ABB RobotStudio station: Assgnt_2_Final.rspag

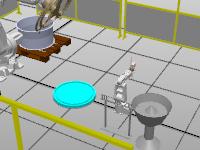
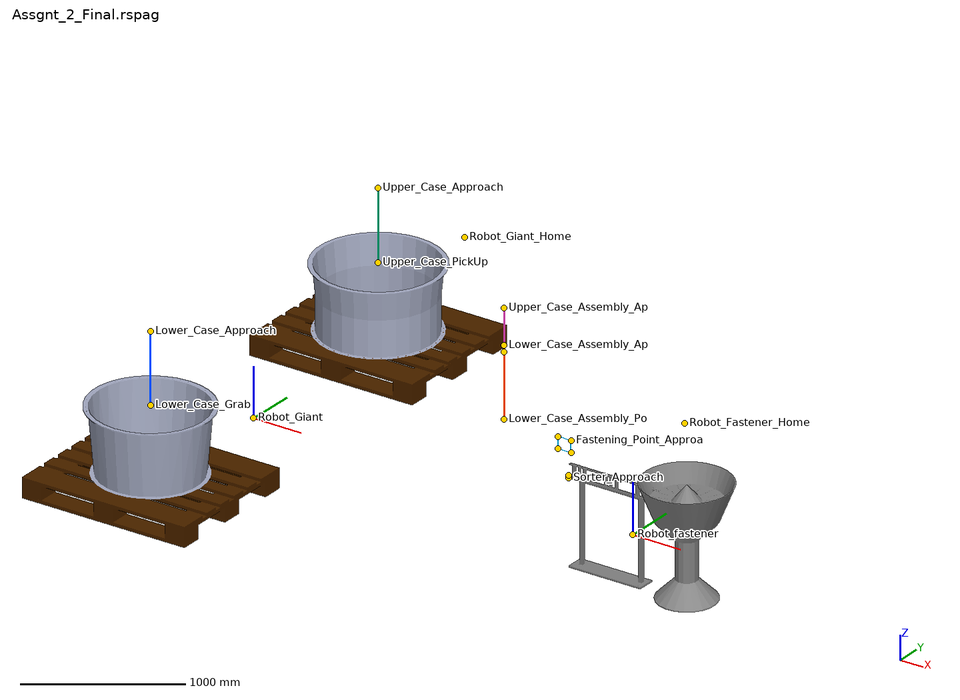
[picture v1: parts stored in the station drawn from their meshes, with robot base, taught points and paths (robot models come from the ABB library and are not in the file)]
--- station ---
Station Assign2_Final (saved by RobotStudio 21.2.9526.0)
Controller Sync_Controller
  mechanical unit ROB_1: Robot_Giant, 6 joints, base frame (0, 0, 0) mm
  mechanical unit ROB_2: Robot_fastener, 6 joints, base frame (2800, 0, 0) mm, rotated rx 0 ry 0 rz 180 deg
Layout (positions relative to the parent item):
  - Robot_Giant [mechanism, from Robots\IRB6620_150_220_G_01.rslib] at (0, 0, 0) mm; joint values [0, 0, 0, 0, 0.5236, 0] (rad or m)
  - UpperEngineCase [part] at (80, 1200, 136) mm, size 855.3 x 860 x 451.6 mm
  - M8_Lock_Nut [part] at (3456.05, -671.29, 653.31) mm, size 15.6 x 13.7 x 11 mm
  - Bolt_nothread [part] at (3473.13, -433.44, 655.7) mm, rotated rx -82.72 ry 0 rz 0 deg, size 20 x 20 x 36 mm
  - Rotating_Base_Mech [mechanism, from Libraries\Rotating_Base_Mech.rslib] at (1850, 0, 0) mm, rotated rx 0 ry 0 rz 37.5 deg; joint values [0] (rad or m)
  - Fence_2500_V1_2 [graphiccomponentgroup, from Equipment\Fence_2500.rslib] at (4110.06, 2559.49, 0) mm, rotated rx 0 ry 0 rz 90 deg
    - Body 1 [part, from Equipment\Fence_2500.rslib]
    - Body 2 [part, from Equipment\Fence_2500.rslib]
  - Fence_2500_H2_2 [graphiccomponentgroup, from Equipment\Fence_2500.rslib] at (-1516.69, -2535.36, 0) mm
    - Body 1 [part, from Equipment\Fence_2500.rslib]
    - Body 2 [part, from Equipment\Fence_2500.rslib]
  - Fence_2500_V1 [graphiccomponentgroup, from Equipment\Fence_2500.rslib] at (1527.78, 2566.59, 0) mm, rotated rx 0 ry 0 rz 90 deg
    - Body 1 [part, from Equipment\Fence_2500.rslib]
    - Body 2 [part, from Equipment\Fence_2500.rslib]
  - Fence_2500_V2 [graphiccomponentgroup, from Equipment\Fence_2500.rslib] at (1521.75, -2665.51, 0) mm, rotated rx 0 ry 0 rz 90 deg
    - Body 1 [part, from Equipment\Fence_2500.rslib]
    - Body 2 [part, from Equipment\Fence_2500.rslib]
  - Fence_2500_H1_2 [graphiccomponentgroup, from Equipment\Fence_2500.rslib] at (4779.67, -2566.91, 0) mm
    - Body 1 [part, from Equipment\Fence_2500.rslib]
    - Body 2 [part, from Equipment\Fence_2500.rslib]
  - Fence_2500_V2_2 [graphiccomponentgroup, from Equipment\Fence_2500.rslib] at (4153.21, -2654.07, 0) mm, rotated rx 0 ry 0 rz 90 deg
    - Body 1 [part, from Equipment\Fence_2500.rslib]
    - Body 2 [part, from Equipment\Fence_2500.rslib]
  - Fence_2500_H1 [graphiccomponentgroup, from Equipment\Fence_2500.rslib] at (4775.16, 0, 0) mm
    - Body 1 [part, from Equipment\Fence_2500.rslib]
    - Body 2 [part, from Equipment\Fence_2500.rslib]
  - Fence_2500_H2 [graphiccomponentgroup, from Equipment\Fence_2500.rslib] at (-1486.79, 0, 0) mm
    - Body 1 [part, from Equipment\Fence_2500.rslib]
    - Body 2 [part, from Equipment\Fence_2500.rslib]
  - Pallet_1 [part] at (80, -1200, 138) mm, rotated rx 90 ry 0 rz 0 deg, size 1200 x 138 x 1000 mm
  - Pallet_2 [part] at (80, 1200, 138) mm, rotated rx 90 ry 0 rz 0 deg, size 1200 x 138 x 1000 mm
  - Robot_fastener [mechanism, from Robots\IRB120_3_58_G_01.rslib] at (2800, 0, 0) mm, rotated rx 0 ry 0 rz 180 deg; joint values [-1.5708, 0, 0, 0, 0, 0] (rad or m)
  - IRC5_Control-Module [part, from Equipment\IRC5_Control-Module.rslib] at (-932.79, 0, 100) mm, rotated rx 90 ry 0 rz 90 deg
  - SC_Grabber [smart component, from Libraries\SC_Grabber.rslib] at (1380.21, 0, 1755) mm, rotated rx 180 ry 60 rz 180 deg
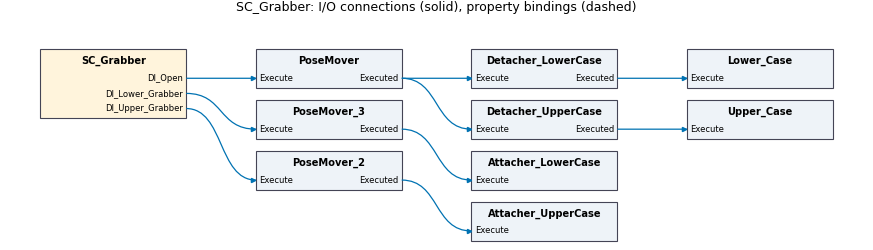
      connections:
        SC_Grabber.DI_Open -> PoseMover.Execute
        SC_Grabber.DI_Lower_Grabber -> PoseMover_3.Execute
        SC_Grabber.DI_Upper_Grabber -> PoseMover_2.Execute
        PoseMover_2.Executed -> Attacher_UpperCase.Execute
        PoseMover_3.Executed -> Attacher_LowerCase.Execute
        PoseMover.Executed -> Detacher_LowerCase.Execute
        PoseMover.Executed -> Detacher_UpperCase.Execute
        Detacher_LowerCase.Executed -> Lower_Case.Execute
        Detacher_UpperCase.Executed -> Upper_Case.Execute
    - Mech_Grabber [mechanism, from Libraries\SC_Grabber.rslib] at (0, 0, 0) mm; joint values [0, 0, 0] (rad or m)
    - PoseMover [smart component, from Components\PoseMover.rslib]
        properties: Mechanism=Mech_Grabber; Pose=2; Duration=0.5
    - PoseMover_2 [smart component, from Components\PoseMover.rslib]
        properties: Mechanism=Mech_Grabber; Pose=3; Duration=0.5
    - PoseMover_3 [smart component, from Components\PoseMover.rslib]
        properties: Mechanism=Mech_Grabber; Pose=4; Duration=0.5
    - Attacher_LowerCase [smart component, from Components\Attacher.rslib]
        properties: Parent=Mech_Grabber; Flange=0; Child=LowerEngineCase; Mount=false; Offset=[0 0 0]; Orientation=[0 0 0]
    - Attacher_UpperCase [smart component, from Components\Attacher.rslib]
        properties: Parent=Mech_Grabber; Flange=0; Child=UpperEngineCase; Mount=false; Offset=[0 0 0]; Orientation=[0 0 0]
    - Detacher_LowerCase [smart component, from Components\Detacher.rslib]
        properties: Child=LowerEngineCase; KeepPosition=true
    - Detacher_UpperCase [smart component, from Components\Detacher.rslib]
        properties: Child=UpperEngineCase; KeepPosition=true
    - Lower_Case [smart component, from Components\SetParent.rslib]
        properties: Child=LowerEngineCase; Parent=Rotating_Base_Mech; KeepTransform=true
    - Upper_Case [smart component, from Components\SetParent.rslib]
        properties: Child=UpperEngineCase; Parent=Rotating_Base_Mech; KeepTransform=true
  - New Nut and Bolt Sorter [part] at (3000, -525, 0) mm, size 1163.5 x 597 x 775 mm
  - SC_Nut_Bolt_Sorter [smart component, from Libraries\SC_Nut_Bolt_Sorter.rslib]
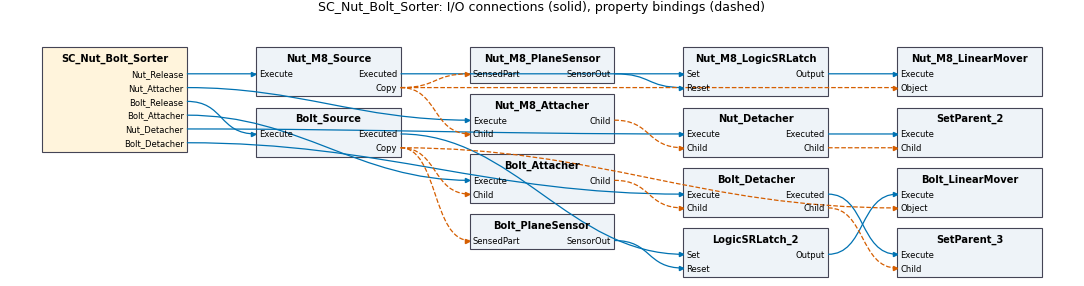
      connections:
        SC_Nut_Bolt_Sorter.Nut_Release -> Nut_M8_Source.Execute
        Nut_M8_Source.Executed -> Nut_M8_LogicSRLatch.Set
        Nut_M8_PlaneSensor.SensorOut -> Nut_M8_LogicSRLatch.Reset
        Nut_M8_LogicSRLatch.Output -> Nut_M8_LinearMover.Execute
        SC_Nut_Bolt_Sorter.Nut_Attacher -> Nut_M8_Attacher.Execute
        SC_Nut_Bolt_Sorter.Bolt_Release -> Bolt_Source.Execute
        Bolt_Source.Executed -> LogicSRLatch_2.Set
        LogicSRLatch_2.Output -> Bolt_LinearMover.Execute
        Bolt_PlaneSensor.SensorOut -> LogicSRLatch_2.Reset
        SC_Nut_Bolt_Sorter.Bolt_Attacher -> Bolt_Attacher.Execute
        SC_Nut_Bolt_Sorter.Nut_Detacher -> Nut_Detacher.Execute
        SC_Nut_Bolt_Sorter.Bolt_Detacher -> Bolt_Detacher.Execute
        Nut_Detacher.Executed -> SetParent_2.Execute
        Bolt_Detacher.Executed -> SetParent_3.Execute
        Nut_M8_Source.Copy => Nut_M8_LinearMover.Object
        Bolt_Source.Copy => Bolt_LinearMover.Object
        Nut_M8_Attacher.Child => Nut_Detacher.Child
        Bolt_Attacher.Child => Bolt_Detacher.Child
        Nut_M8_Source.Copy => Nut_M8_PlaneSensor.SensedPart
        Bolt_Source.Copy => Bolt_PlaneSensor.SensedPart
        Nut_M8_Source.Copy => Nut_M8_Attacher.Child
        Bolt_Source.Copy => Bolt_Attacher.Child
        Nut_Detacher.Child => SetParent_2.Child
        Bolt_Detacher.Child => SetParent_3.Child
    - Nut_M8_Source [smart component, from Components\Source.rslib]
        properties: Source=M8_Lock_Nut; Copy=(none); Parent=(none); Position=[3.340616 -0.525502 0.575]; Orientation=[0 0 0]; Transient=false; PhysicsBehavior=0
    - Nut_M8_LogicSRLatch [smart component, from Components\LogicSRLatch.rslib]
    - Nut_M8_PlaneSensor [smart component, from Components\PlaneSensor.rslib]
        properties: Origin=[2.69 -0.58 0.55]; Axis1=[0 0.1 0]; Axis2=[0 0 0.06]; SensedPart=(none)
      - _sensorPart_ [part, from Libraries\SC_Nut_Bolt_Sorter.rslib]
    - Nut_M8_LinearMover [smart component, from Components\LinearMover.rslib]
        properties: Object=(none); Direction=[-0.64172 0 0]; Speed=0.3; Reference=Global; ReferenceObject=(none)
    - Nut_M8_Attacher [smart component, from Components\Attacher.rslib]
        properties: Parent=SC_Fastener_New; Flange=0; Child=(none); Mount=false; Offset=[0 0 0]; Orientation=[0 0 0]
    - Bolt_Attacher [smart component, from Components\Attacher.rslib]
        properties: Parent=SC_Fastener_New; Flange=0; Child=(none); Mount=false; Offset=[0 0 0]; Orientation=[0 0 0]
    - Bolt_LinearMover [smart component, from Components\LinearMover.rslib]
        properties: Object=(none); Direction=[-1 0 0]; Speed=0.3; Reference=Global; ReferenceObject=(none)
    - Bolt_PlaneSensor [smart component, from Components\PlaneSensor.rslib]
        properties: Origin=[2.69 -0.58 0.65]; Axis1=[0 0.1 0]; Axis2=[0 0 0.06]; SensedPart=(none)
      - _sensorPart_ [part, from Libraries\SC_Nut_Bolt_Sorter.rslib]
    - LogicSRLatch_2 [smart component, from Components\LogicSRLatch.rslib]
    - Bolt_Source [smart component, from Components\Source.rslib]
        properties: Source=Bolt_nothread; Copy=(none); Parent=(none); Position=[3.306216 -0.525502 0.64]; Orientation=[0 0 0]; Transient=false; PhysicsBehavior=0
    - Nut_Detacher [smart component, from Components\Detacher.rslib]
        properties: Child=(none); KeepPosition=true
    - Bolt_Detacher [smart component, from Components\Detacher.rslib]
        properties: Child=(none); KeepPosition=true
    - SetParent_2 [smart component, from Components\SetParent.rslib]
        properties: Child=(none); Parent=Rotating_Base_Mech; KeepTransform=true
    - SetParent_3 [smart component, from Components\SetParent.rslib]
        properties: Child=(none); Parent=Rotating_Base_Mech; KeepTransform=true
  - LowerEngineCase [part] at (80, -1200, 136) mm, size 821.5 x 826 x 454 mm
  - SC_Fastener_New [smart component, from Libraries\SC_Fastener_New.rslib] at (2800, 374, 630) mm, rotated rx 0 ry 90 rz 90 deg
      connections:
        SC_Fastener_New.FNDI_Home -> PoseMover.Execute
        SC_Fastener_New.FNDI_Open -> PoseMover_2.Execute
        SC_Fastener_New.FNDI_ClosePick -> PoseMover_3.Execute
    - Mech_Fastening_New [mechanism, from Libraries\SC_Fastener_New.rslib] at (0, 0, 0) mm; joint values [-0.07, 0.0705] (rad or m)
    - PoseMover [smart component, from Components\PoseMover.rslib]
        properties: Mechanism=Mech_Fastening_New; Pose=1; Duration=0.5
    - PoseMover_2 [smart component, from Components\PoseMover.rslib]
        properties: Mechanism=Mech_Fastening_New; Pose=2; Duration=0.5
    - PoseMover_3 [smart component, from Components\PoseMover.rslib]
        properties: Mechanism=Mech_Fastening_New; Pose=3; Duration=0.5
  - SC_Rotate_Base [smart component, from Libraries\SC_Rotate_Base.rslib]
      connections:
        SC_Rotate_Base.DI_Rotate -> Base.Execute
    - Base [smart component, from Components\Rotator2.rslib]
        properties: Object=Rotating_Base_Mech; CenterPoint=[0 0 0]; Axis=[0 0 0.001]; Angle=0.130899693899575; Duration=1; Reference=Local; ReferenceObject=(none)
Attachment: SC_Grabber is attached to Robot_Giant / Link6
Attachment: SC_Fastener_New is attached to Robot_fastener / Link6
Station signals: DI Trail_Breaker
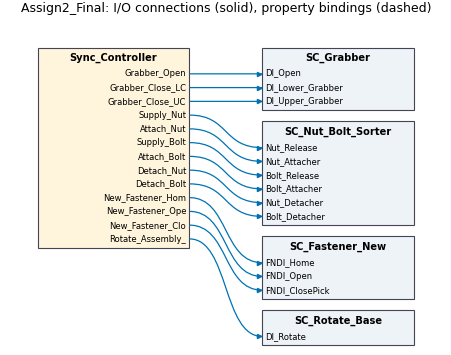
Station logic (signal -> signal, property => property):
  Sync_Controller.Grabber_Open -> SC_Grabber.DI_Open
  Sync_Controller.Grabber_Close_LC -> SC_Grabber.DI_Lower_Grabber
  Sync_Controller.Grabber_Close_UC -> SC_Grabber.DI_Upper_Grabber
  Sync_Controller.Supply_Nut -> SC_Nut_Bolt_Sorter.Nut_Release
  Sync_Controller.Attach_Nut -> SC_Nut_Bolt_Sorter.Nut_Attacher
  Sync_Controller.Supply_Bolt -> SC_Nut_Bolt_Sorter.Bolt_Release
  Sync_Controller.Attach_Bolt -> SC_Nut_Bolt_Sorter.Bolt_Attacher
  Sync_Controller.Detach_Nut -> SC_Nut_Bolt_Sorter.Nut_Detacher
  Sync_Controller.Detach_Bolt -> SC_Nut_Bolt_Sorter.Bolt_Detacher
  Sync_Controller.New_Fastener_Home -> SC_Fastener_New.FNDI_Home
  Sync_Controller.New_Fastener_Open -> SC_Fastener_New.FNDI_Open
  Sync_Controller.New_Fastener_ClosePick -> SC_Fastener_New.FNDI_ClosePick
  Sync_Controller.Rotate_Assembly_Base -> SC_Rotate_Base.DI_Rotate

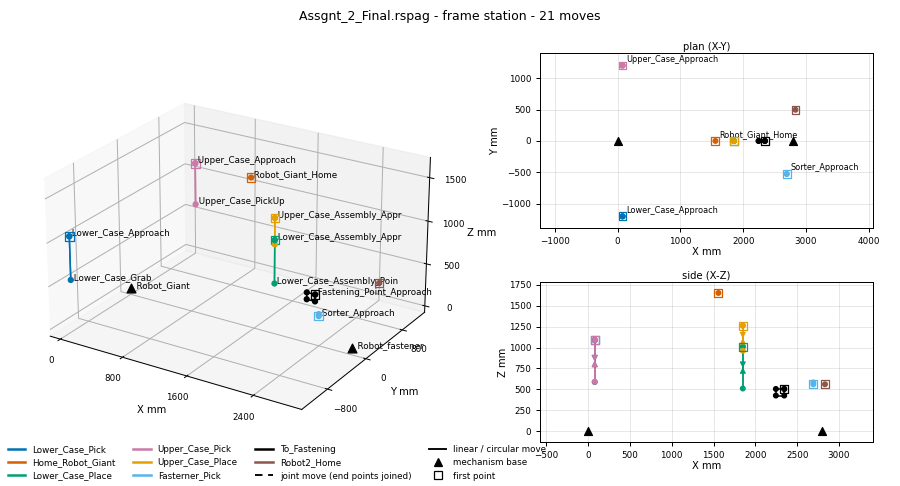
[picture p0: tool path of Assgnt_2_Final.rspag in frame station, 21 of 21 moves have a stored position in this frame; points joined in program order, loops and branches not executed]
--- Backups/Sync_Controller/RAPID/TASK1/PROGMOD/CalibData.mod ---
MODULE CalibData
    PERS tooldata Mech_Grabber_1:=[TRUE,[[0,0,205.5],[1,0,0,0]],[2,[0,0,200],[1,0,0,0],0,0,0]];
    TASK PERS wobjdata Wobj_Lower_Case:=[FALSE,TRUE,"",[[80.0405,-1200,592],[0.999974,-0.00506277,0.00506303,0.000025634]],[[0,0,0],[1,0,0,0]]];
    TASK PERS wobjdata Wobj_Upper_Case:=[FALSE,TRUE,"",[[80,1200,589.619],[1,0,0,0]],[[0,0,0],[1,0,0,0]]];
    TASK PERS wobjdata Wobj_Assembly:=[FALSE,TRUE,"",[[1850,0,60],[1,0,0,0]],[[0,0,0],[1,0,0,0]]];
ENDMODULE

--- Backups/Sync_Controller/RAPID/TASK1/PROGMOD/Module1.mod ---
MODULE Module1
        CONST robtarget Lower_Case_Approach:=[[-5.063031994,-5.022012339,495.949144175],[-0.000000184,0.707106781,0.707070529,0.007160025],[0,0,0,0],[9E+09,9E+09,9E+09,9E+09,9E+09,9E+09]];
    CONST robtarget Lower_Case_Grab:=[[0.000000003,0.0405001,-3.999589872],[0.000000184,0.707106781,0.707070529,0.007160025],[0,0,0,0],[9E+09,9E+09,9E+09,9E+09,9E+09,9E+09]];
    CONST robtarget Robot_Giant_Home:=[[1558.173301235,0,1652.25],[0.5,0,0.866025404,0],[0,0,0,0],[9E+09,9E+09,9E+09,9E+09,9E+09,9E+09]];
    CONST robtarget Lower_Case_Assembly_Approach:=[[0,0,950],[0,0,1,0],[0,0,0,0],[9E+09,9E+09,9E+09,9E+09,9E+09,9E+09]];
    CONST robtarget Lower_Case_Assembly_Point:=[[0,0,450],[0,0,1,0],[0,0,0,0],[9E+09,9E+09,9E+09,9E+09,9E+09,9E+09]];
    CONST robtarget Upper_Case_Approach:=[[0,0,500],[0,-0.707106779,0.707106783,-0.000000368],[0,0,0,0],[9E+09,9E+09,9E+09,9E+09,9E+09,9E+09]];
    CONST robtarget Upper_Case_PickUp:=[[0,0,0],[0,-0.707106779,0.707106783,-0.000000368],[0,-1,-1,0],[9E+09,9E+09,9E+09,9E+09,9E+09,9E+09]];
    CONST robtarget Upper_Case_Assembly_Approach:=[[0,0,1201.62],[0,0,1,0],[0,0,0,0],[9E+09,9E+09,9E+09,9E+09,9E+09,9E+09]];
    CONST robtarget Upper_Case_Assembly_Point:=[[0,0,901.62],[0,0,1,0],[0,0,0,0],[9E+09,9E+09,9E+09,9E+09,9E+09,9E+09]];
!***********************************************************
    !
    ! Module:  Module1
    !
    ! Description:
    !   <Insert description here>
    !
    ! Author: Santosh Govindaraj
    !
    ! Version: 1.0
    !
    !***********************************************************


    !***********************************************************
    !
    ! Procedure main
    !
    !   This is the entry point of your program
    !
    !***********************************************************
    PROC main()
        !Add your code here
        Home_Robot_Giant;
        Lower_Case_Pick;
        Lower_Case_Place;
        Upper_Case_Pick;
        Upper_Case_Place;
        Home_Robot_Giant;
    ENDPROC
    PROC Lower_Case_Pick()
        SetDO Grabber_Open,1;
        SetDO Grabber_Close_LC,0;
        MoveL Lower_Case_Approach,v1000,z100,Mech_Grabber_1\WObj:=Wobj_Lower_Case;
        MoveL Lower_Case_Grab,v1000,z100,Mech_Grabber_1\WObj:=Wobj_Lower_Case;
        WaitTime 0.5;
        SetDO Grabber_Open,0;
        SetDO Grabber_Close_LC,1;
        WaitTime 1;
        MoveL Lower_Case_Approach,v1000,z100,Mech_Grabber_1\WObj:=Wobj_Lower_Case;
    ENDPROC
    PROC MAIN_ROB1()
        Home_Robot_Giant;
        Lower_Case_Pick;
        Lower_Case_Place;
        Upper_Case_Pick;
        Upper_Case_Place;
        Home_Robot_Giant;
    ENDPROC
    PROC Home_Robot_Giant()
        MoveL Robot_Giant_Home,v1000,z100,Mech_Grabber_1\WObj:=wobj0;
    ENDPROC
    PROC Lower_Case_Place()
        MoveL Lower_Case_Assembly_Approach,v1000,z100,Mech_Grabber_1\WObj:=Wobj_Assembly;
        MoveL Lower_Case_Assembly_Point,v1000,z100,Mech_Grabber_1\WObj:=Wobj_Assembly;
        SetDO Grabber_Close_LC,0;
        WaitTime 1;
        SetDO Grabber_Open,1;
        SetDO Grabber_Open,0;
        WaitTime 1;
        MoveL Lower_Case_Assembly_Approach,v1000,z100,Mech_Grabber_1\WObj:=Wobj_Assembly;
    ENDPROC
    PROC Upper_Case_Pick()
        SetDO Grabber_Open,1;
        SetDO Grabber_Close_UC,0;
        SetDO Grabber_Open,0;
        MoveL Upper_Case_Approach,v1000,z100,Mech_Grabber_1\WObj:=Wobj_Upper_Case;
        MoveL Upper_Case_PickUp,v1000,z100,Mech_Grabber_1\WObj:=Wobj_Upper_Case;
        WaitTime 0.5;
        SetDO Grabber_Close_UC,1;
        WaitTime 1;
        MoveL Upper_Case_Approach,v1000,z100,Mech_Grabber_1\WObj:=Wobj_Upper_Case;
    ENDPROC
    PROC Upper_Case_Place()
        MoveL Upper_Case_Assembly_Approach,v1000,z100,Mech_Grabber_1\WObj:=Wobj_Assembly;
        MoveL Upper_Case_Assembly_Point,v1000,z100,Mech_Grabber_1\WObj:=Wobj_Assembly;
        SetDO Grabber_Close_UC,0;
        WaitTime 1;
        SetDO Grabber_Open,1;
        SetDO Grabber_Open,0;
        WaitTime 1;
        MoveL Upper_Case_Assembly_Approach,v1000,z100,Mech_Grabber_1\WObj:=Wobj_Assembly;
    ENDPROC
    PROC Path_10()

    ENDPROC
    PROC ROBOT()
        Home_Robot_Giant;
        Lower_Case_Pick;
        Lower_Case_Place;
        Upper_Case_Pick;
        Upper_Case_Place;
        Home_Robot_Giant;
    ENDPROC
ENDMODULE

--- Backups/Sync_Controller/RAPID/TASK2/PROGMOD/CalibData.mod ---
MODULE CalibData
    PERS tooldata Mech_Fastener_1:=[TRUE,[[-12,-31.5,121],[1,0,0,0]],[1,[0.1,0,0],[1,0,0,0],0,0,0]];
    PERS tooldata Mech_Fastner_1:=[TRUE,[[69,-32,122],[0.707107,0,0.707107,0]],[1.5,[0.1,0,0],[1,0,0,0],0,0,0]];
    TASK PERS wobjdata Wobj_Sorter:=[FALSE,TRUE,"",[[2699.22,-537.502,584],[1,0,0,0]],[[0,0,0],[1,0,0,0]]];
    TASK PERS wobjdata Wobj_Fastening:=[FALSE,TRUE,"",[[1850,0,60],[1,0,0,0]],[[0,0,0],[1,0,0,0]]];
    PERS tooldata Mech_Fastening_New_1:=[TRUE,[[139.999,-31.395,121.281],[0.707107,0,0.707107,0]],[2,[50,50,50],[1,0,0,0],0,0,0]];
ENDMODULE

--- Backups/Sync_Controller/RAPID/TASK2/PROGMOD/Module1.mod ---
MODULE Module1
        CONST robtarget Target_10:=[[2831.999489549,496.000032596,560.999998333],[0.000000002,0.707107145,-0.707106417,0.000000002],[-1,0,-1,0],[9E+09,9E+09,9E+09,9E+09,9E+09,9E+09]];
    CONST robtarget Target_20:=[[2742.402,-523,589.664],[0.000000002,0.707106417,0.707107145,0.000000002],[0,-2,1,1],[9E+09,9E+09,9E+09,9E+09,9E+09,9E+09]];
    CONST robtarget Target_30:=[[2745.508,-494.542,588.187],[0.000000002,0.707106417,0.707107145,0.000000002],[0,-2,1,1],[9E+09,9E+09,9E+09,9E+09,9E+09,9E+09]];
    CONST robtarget Bolt_attac:=[[2745.875,-494.542,676],[0.000000002,0.707106417,0.707107145,0.000000002],[0,0,-1,0],[9E+09,9E+09,9E+09,9E+09,9E+09,9E+09]];
    CONST robtarget Sorter_Approach:=[[-6.6,12,-24],[0,0.707106781,0.707106781,0],[0,0,-1,0],[9E+09,9E+09,9E+09,9E+09,9E+09,9E+09]];
    CONST robtarget Sorter_Pick:=[[-6.6,12,-2],[0,0.707106781,0.707106781,0],[0,0,-1,0],[9E+09,9E+09,9E+09,9E+09,9E+09,9E+09]];
    CONST robtarget Fastening_Point_Approach:=[[495,0,445],[0,1,0,0],[0,-2,1,0],[9E+09,9E+09,9E+09,9E+09,9E+09,9E+09]];
    CONST robtarget Fastening_Point:=[[395,0,445],[0,1,0,0],[0,-2,1,0],[9E+09,9E+09,9E+09,9E+09,9E+09,9E+09]];
    CONST robtarget Robot_Fastener_Home:=[[2831.999489549,496.000032596,560.999998333],[0.000000002,0.707107145,-0.707106417,0.000000002],[-1,0,-1,0],[9E+09,9E+09,9E+09,9E+09,9E+09,9E+09]];
    CONST robtarget Fastening_Point_Down:=[[395,0,366],[0,1,0,0],[0,-2,1,0],[9E+09,9E+09,9E+09,9E+09,9E+09,9E+09]];
    CONST robtarget Fastening_Wait_For_Next:=[[495,0,366],[0,1,0,0],[0,-2,1,0],[9E+09,9E+09,9E+09,9E+09,9E+09,9E+09]];
!***********************************************************
    !
    ! Module:  Module1
    !
    ! Description:
    !   <Insert description here>
    !
    ! Author: Santosh Govindaraj
    !
    ! Version: 1.0
    !
    !***********************************************************


    !***********************************************************
    !
    ! Procedure main
    !
    !   This is the entry point of your program
    !
    !***********************************************************
    PROC main()
        !Add your code here
    ENDPROC
    PROC Suppliers()
        SetDO Supply_Nut,0;
        SetDO Supply_Bolt,0;
        WaitTime 0.5;
        SetDO Supply_Nut,1;
        SetDO Supply_Bolt,1;
        WaitTime 1;
    ENDPROC
    PROC Robot2_Task()
        SetDO New_Fastener_Home,0;
        WaitTime 18;
        Robot2_Home;
        FOR loop FROM 0 TO 47 DO
            Fasten_And_Rotate;
        ENDFOR
        Robot2_Home;
    ENDPROC
    PROC Fasterner_Pick()
        SetDO New_Fastener_Open,1;
        SetDO New_Fastener_Open,0;
        SetDO Attach_Nut,0;
        SetDO Attach_Bolt,0;
        WaitTime 0.5;
        MoveJ Sorter_Approach,v2000,fine,Mech_Fastening_New_1\WObj:=Wobj_Sorter;
        MoveL Sorter_Pick,v1000,fine,Mech_Fastening_New_1\WObj:=Wobj_Sorter;
        SetDO Attach_Nut,1;
        SetDO New_Fastener_ClosePick,1;
        WaitTime 0.5;
        SetDO New_Fastener_ClosePick,0;
        SetDO Attach_Bolt,1;
        WaitTime 0.5;
        SetDO Attach_Nut,0;
        SetDO Attach_Bolt,0;
    ENDPROC
    PROC To_Fastening()
        MoveJ Fastening_Point_Approach,v1000,fine,Mech_Fastening_New_1\WObj:=Wobj_Fastening;
        MoveJ Fastening_Point,v500,fine,Mech_Fastening_New_1\WObj:=Wobj_Fastening;
        WaitTime 0.5;
        SetDO Detach_Nut,1;
        SetDO New_Fastener_Home,0;
        WaitTime 0.5;
        SetDO New_Fastener_Home,1;
        MoveL Fastening_Point_Down,v500,fine,Mech_Fastening_New_1\WObj:=Wobj_Fastening;
        WaitTime 0.2;
        SetDO Detach_Bolt,1;
        WaitTime 0.5;
        SetDO Detach_Bolt,0;
        SetDO Detach_Nut,0;
        SetDO New_Fastener_Open,1;
        WaitTime 0.2;
        SetDO New_Fastener_Open,0;
        MoveL Fastening_Wait_For_Next,v1000,fine,Mech_Fastening_New_1\WObj:=Wobj_Fastening;
        MoveJ Fastening_Point_Approach,v1000,fine,Mech_Fastening_New_1\WObj:=Wobj_Fastening;
    ENDPROC
    PROC Robot2_Home()
        MoveJ Robot_Fastener_Home,v2000,fine,Mech_Fastner_1\WObj:=wobj0;
    ENDPROC
    PROC Fasten_And_Rotate()
        Suppliers;
        WaitTime .5;
        Fasterner_Pick;
        To_Fastening;
        SetDO Rotate_Assembly_Base,0;
        WaitTime 0.5;
        SetDO Rotate_Assembly_Base,1;
    ENDPROC
ENDMODULE

--- Backups/Sync_Controller/SYSPAR/EIO.cfg ---
EIO:CFG_1.0:6:1::
#
EIO_SIGNAL:

      -Name "Grabber_Open" -SignalType "DO" -Access "All"

      -Name "Grabber_Close_LC" -SignalType "DO" -Access "All"

      -Name "Grabber_Close_UC" -SignalType "DO" -Access "All"

      -Name "Supply_Nut" -SignalType "DO" -Access "All"

      -Name "Attach_Nut" -SignalType "DO" -Access "All"

      -Name "Attach_Bolt" -SignalType "DO" -Access "All"

      -Name "Supply_Bolt" -SignalType "DO" -Access "All"

      -Name "Detach_Nut" -SignalType "DO" -Access "All"

      -Name "Detach_Bolt" -SignalType "DO" -Access "All"

      -Name "New_Fastener_Home" -SignalType "DO" -Access "All"

      -Name "New_Fastener_Open" -SignalType "DO" -Access "All"

      -Name "New_Fastener_ClosePick" -SignalType "DO" -Access "All"

      -Name "Rotate_Assembly_Base" -SignalType "DO" -Access "All"
